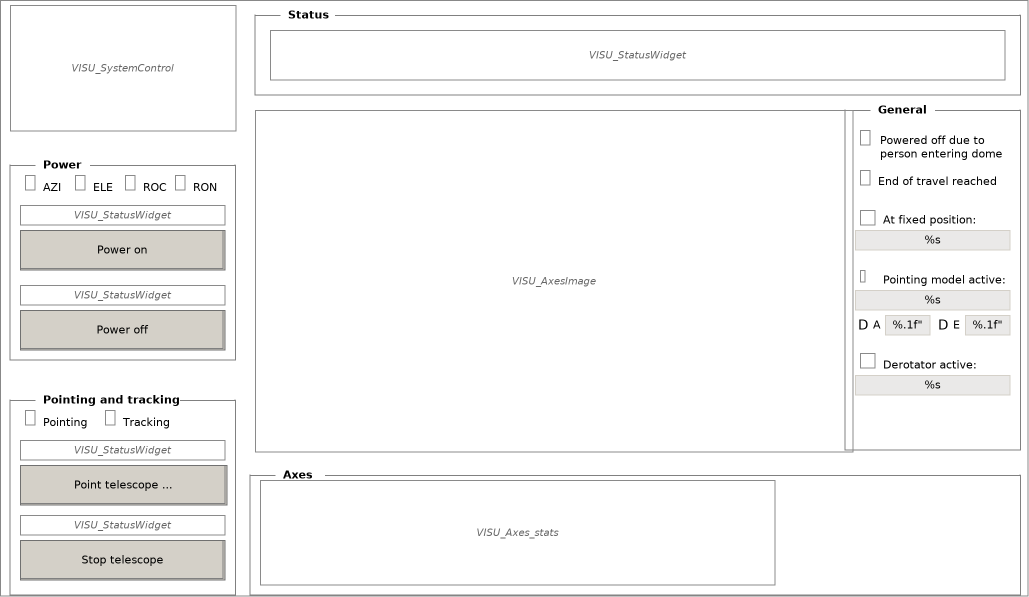
VISUALIZATION VISU_AxesOverview  // 1029x597
VAR_IN_OUT
	ref : Axes;
    widget : AxesWidget;
END_VAR
    Polyline (935,110) (1020,110) (1020,450) (845,450) (845,110) (870,110)
    Frame (255,110 598x342)
        shows VISU_AxesImage(ref := ref, widget := widget)
    Polyline (180,400) (235,400) (235,595) (10,595) (10,400) (35,400)
    Polyline (90,165) (235,165) (235,360) (10,360) (10,165) (35,165)
    Frame (10,5 226x126)
        shows VISU_SystemControl(status := widget.actualStatus, button_initialize := widget.button_initialize, button_operating := widget.button_operating, button_locking := widget.button_locking)
    Button (20,230 205x40), "Power on", input disabled if: ref.processes.powerOn.statuses.enabledStatus.disabled
        OnMouseClick: execute {
            ref.processes.powerOn.request(
                azi := TRUE,
                ele := TRUE,
                roc := FALSE,
                ron := FALSE,
                fw := FALSE);
        }
    Button (20,540 205x40), "Stop telescope", input disabled if: ref.processes.stop.statuses.enabledStatus.disabled
        OnMouseClick: execute { ref.processes.stop.do_request := TRUE; }
    Button (20,310 205x40), "Power off", input disabled if: ref.processes.powerOff.statuses.enabledStatus.disabled
        OnMouseClick: execute { ref.processes.powerOff.do_request := TRUE; }
    Frame (25,175 10x15)
        shows VISU_State_gray_green(state := ref.parts.azi.statuses.poweredStatus.enabled)
    Label (40,175 30x25), "AZI"
    Button (20,465 207x40), "Point telescope ..."
        OnMouseClick: OpenDialog Dialog=VISU_AxesPointDialog, OpenModal=True, OpenCentered=True
    Frame (860,130 10x15)
        shows VISU_State_gray_orange(state := ref.isPoweredOffByPersonInDome)
    Label (877,132 150x30), "Powered off due to person entering dome"
    Rectangle (855,230 155x20), "%s", text variable: ref.actualKnownPositionName, colour toggle: ref.isAtKnownPosition
    Label (880,205 125x30), "At fixed position:"
    Rectangle (855,290 155x20), "%s", text variable: widget.activePointingModelString
    Label (880,265 140x30), "Pointing model active:"
    Rectangle (855,375 155x20), "%s", text variable: widget.activeRotatorString
    Label (880,355 125x20), "Derotator active:"
    Label (40,155 50x20), "Power"
    Frame (20,515 205x20)
        shows VISU_StatusWidget(widget := widget.processes_stopStatus)
        p4168582468: ref.processes.stop.actualStatus
    Frame (20,440 205x20)
        shows VISU_StatusWidget(widget := widget.processes_pointStatus)
        p4168582468: ref.processes.point.actualStatus
    Frame (20,285 205x20)
        shows VISU_StatusWidget(widget := widget.processes_powerOffStatus)
        p4168582468: ref.processes.reset.actualStatus
    Frame (20,205 205x20)
        shows VISU_StatusWidget(widget := widget.processes_powerOnStatus)
        p4168582468: ref.processes.reset.actualStatus
    Label (40,390 135x20), "Pointing and tracking"
    Frame (75,175 10x15)
        shows VISU_State_gray_green(state := ref.parts.ele.statuses.poweredStatus.enabled)
    Label (90,175 30x25), "ELE"
    Frame (125,175 10x15)
        shows VISU_State_gray_green(state := ref.parts.roc.statuses.poweredStatus.enabled)
    Label (140,175 30x25), "ROC"
    Frame (175,175 10x15)
        shows VISU_State_gray_green(state := ref.parts.ron.statuses.poweredStatus.enabled)
    Label (190,175 30x25), "RON"
    Frame (25,410 10x15)
        shows VISU_State_gray_green(state := ref.isPointing)
    Label (40,410 60x25), "Pointing"
    Label (120,410 60x25), "Tracking"
    Frame (105,410 10x15)
        shows VISU_State_gray_green(state := ref.isTracking)
    Frame (860,270 5x12)
        shows VISU_State_red_green(state := ref.isPointingModelActive)
    Frame (860,210 15x15)
        shows VISU_State_gray_green(state := ref.isAtKnownPosition)
    Frame (860,353 15x15)
        shows VISU_State_gray_green(state := widget.isDerotatorActive)
    Label (870,315 15x20), "A"
    Label (855,315 20x20), "D"
    Rectangle (885,315 45x20), "%.1f"", text variable: ref.target.aziPointingModelOffset.arcseconds.value
    Label (950,315 15x20), "E"
    Label (935,315 20x20), "D"
    Rectangle (965,315 45x20), "%.1f"", text variable: ref.target.elePointingModelOffset.arcseconds.value
    Frame (860,170 10x15)
        shows VISU_State_gray_red(state := ref.isLimitsReached)
    Label (875,170 150x23), "End of travel reached"
    Polyline (335,15) (1020,15) (1020,95) (255,95) (255,15) (280,15)
    Label (285,5 50x20), "Status"
    Frame (270,30 735x50)
        shows VISU_StatusWidget(widget := widget.actualStatus)
        p4168582468: ref.processes.reset.actualStatus
    Polyline (325,475) (1020,475) (1020,595) (250,595) (250,475) (275,475)
    Label (280,465 70x20), "Axes"
    Frame (260,480 515x105)
        shows VISU_Axes_stats(ref := ref, widget := widget)
    Label (875,100 70x20), "General"
END_VISUALIZATION

(* stored: Version 1.1.0.1, ProductVersion 3.1.4019.2
   Visu VISU_AxesOverview: Id {cd72824b-3f00-476e-8415-7fec96d83dec} *)
